FUNCTION_BLOCK FB_StringBuilder

VAR
	{attribute 'hide'}
	_dataBuffer		: ARRAY[0..MaxBufferSize] OF BYTE;  // Buffer for storing of all text
	_dataBufferAdd 	: POINTER TO BYTE; // Databuffer start adress
	_currentLength 	: UDINT; // Current length of string in databuffer. 
END_VAR

VAR CONSTANT
	MaxBufferSize : UDINT := 49999999; // max 50MB buffer 	
END_VAR

METHOD Append : BOOL
VAR_INPUT
	InputString : T_MaxString;
END_VAR
VAR
	StringLength: UDINT;
END_VAR

StringLength := DINT_TO_UDINT(LEN(InputString));
Append := THIS^.AppendGeneric(ADR(InputString),StringLength);
END_METHOD

METHOD AppendGeneric : BOOL
VAR_INPUT
	AddressPointer : POINTER TO BYTE; // Pointer to data
	DataLength : UDINT; 
END_VAR
IF _dataBufferAdd = 0 THEN
	_dataBufferAdd := ADR(_dataBuffer);
END_IF

IF _currentLength + DataLength < MaxBufferSize AND DataLength > 0 THEN
	MEMCPY(_dataBufferAdd + _currentLength, AddressPointer, DataLength);
	_currentLength := _currentLength + DataLength;
	AppendGeneric := TRUE;
ELSE
	AppendGeneric := FALSE;
END_IF
END_METHOD

METHOD AppendLine : BOOL
VAR_INPUT
	InputString : T_MaxString;
END_VAR
THIS^.Append(InputString);
THIS^.Append('$R$N');
END_METHOD

PROPERTY BufferSize : UDINT
GET
BufferSize := MaxBufferSize;
END_GET
END_PROPERTY

METHOD Clear : BOOL
VAR_INPUT
END_VAR
_currentLength := 0;
END_METHOD

METHOD GetIndexOf : DINT
VAR_INPUT
	SearchString	: T_MAXSTRING; 
	StartIndex		: UDINT;
END_VAR
VAR
	searchStringLength : UDINT;
	
	iStringIndex	: UDINT;

	
	matchFound 	: BOOL;

	

 
END_VAR



searchStringLength := TO_UDINT(LEN(SearchString));

IF StartIndex < 0 THEN
	StartIndex := 0;
END_IF

matchFound := FALSE; 
IF (searchStringLength <= THIS^.Length) AND (StartIndex <  THIS^.Length-searchStringLength) THEN
	FOR iStringIndex := StartIndex TO (THIS^.Length-searchStringLength) DO
		// Loop through current string.
	
		
		// Search for string
		
		matchFound := memcmp(	pBuf1 	:= THIS^.StringPointer + iStringIndex,
								pBuf2 	:= ADR(SearchString),
								n		:= searchStringLength) = 0;  
	
	
		IF matchFound THEN
			EXIT;
		END_IF
	END_FOR
END_IF
IF matchFound THEN
	GetIndexOf := TO_DINT(iStringIndex); 
ELSE
	GetIndexOf := -1;
END_IF
END_METHOD

METHOD Initialize : BOOL
IF _dataBufferAdd = 0 THEN
	_dataBufferAdd := ADR(_dataBuffer);
END_IF
END_METHOD

PROPERTY Length : UDINT
GET
Length := _currentLength;
END_GET
SET
_currentLength := Length;
END_SET
END_PROPERTY

PROPERTY StringPointer : POINTER TO BYTE
GET
StringPointer := _dataBufferAdd;
END_GET
END_PROPERTY

PROPERTY ToString : STRING(255)
GET
VAR_INST
	s255String : STRING(255);
	length : UDINT;
END_VAR
s255String := '';
length := MIN(_currentLength, DINT_TO_UDINT(SIZEOF(s255String)));
MEMCPY(ADR(s255String), _dataBufferAdd, length);
ToString := s255String;
END_GET
END_PROPERTY

PROPERTY ToStringEnding : STRING(255)
GET
VAR_INST
	s255String : STRING(255);
	length : UDINT;
END_VAR
s255String := '';
length := 255;
IF _currentLength > 255 THEN
	MEMCPY(ADR(s255String), _dataBufferAdd+_currentLength-length, length);
ELSE
	s255String := 'Length less than 255'; 
END_IF
ToStringEnding := s255String;
END_GET
END_PROPERTY

END_FUNCTION_BLOCK

(* stored: Version 1.1.0.1, ProductVersion 3.1.4022.11
   POU FB_StringBuilder: Id {dee2e3a7-bc35-4e5e-a9ca-fb16e4ba4746}, SpecialFunc None
   Method Append: Id {f0a312ae-549f-4e90-b105-c9135daa53e1}
   Method AppendGeneric: Id {4a606af7-0130-4cd1-a940-87be6db83117}
   Method AppendLine: Id {ac2956bf-22dc-44c9-a789-21f1b2ed884d}
   Property BufferSize: Id {346c3946-c687-4e0b-9485-e2b9636c0948}
   Get Get: Id {d1c51689-53e3-4ce3-8080-77330e73e4f9}
   Method Clear: Id {9f431463-da2d-4510-8a8b-f04590f59e86}
   Method GetIndexOf: Id {6091a517-dfa1-4c73-9dd3-c93c50c8e7a5}
   Method Initialize: Id {b99fed44-03f1-496f-bfcf-4437aa3bee38}
   Property Length: Id {f9ab0fc7-6034-4372-87d7-8ead9a6e691c}
   Get Get: Id {a4200f6c-b58b-48e1-857f-aee972d8d68f}
   Set Set: Id {bfa0876b-e475-4546-b2fd-c73f093a74a2}
   Property StringPointer: Id {d30c913a-63ac-4fce-87e4-9296bb47ba86}
   Get Get: Id {b0463481-0e33-474a-b2b0-403f089bbd65}
   Property ToString: Id {14c21fa1-a7bc-4c30-9754-002c8e4f7e18}
   Get Get: Id {338ff9f4-6df7-4e86-b701-a5f1f679b1dc}
   Property ToStringEnding: Id {361709f6-d66f-443b-9ed2-65397681654c}
   Get Get: Id {878ee556-cb6b-4d13-a15c-724360e2c0ed} *)
